// LS Electric XG5000 project: day27
// PLC LSPLC
// module base 0 slot 0: 입출력 모듈:XBC-DR30S (DC 24V 입력 18점, 릴레이 출력 12점)

PROGRAM day27 (task: 스캔 프로그램)

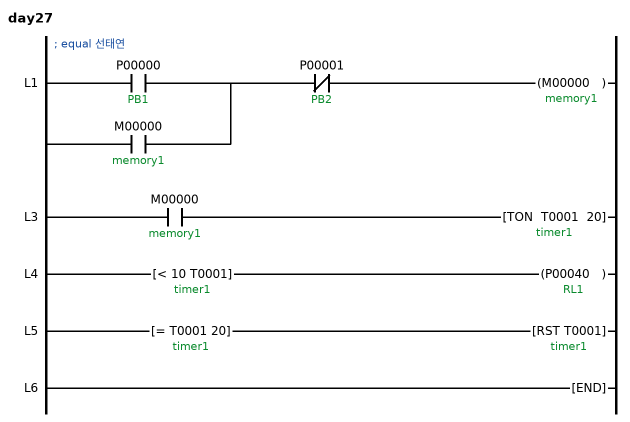
// equal 선태연
; L1
LOAD      P00000	// PB1
OR        M00000	// memory1
AND NOT   P00001	// PB2
OUT       M00000	// memory1
; L3
LOAD      M00000	// memory1
TON       T0001 20	// timer1
; L4
LOAD<     10 T0001	// timer1
OUT       P00040	// RL1
; L5
LOAD=     T0001 20	// timer1
RST       T0001	// timer1
; L6
END